PROGRAM Callblocks
VAR
	
Temp_bool : BOOL;
Mode_0          : Mode;
Feedback_FD     : Feedback_FB;
Feedback_RD     : Feedback_FB;
Feedback_FX1TR  : Feedback_FB;
Feedback_FX2TR  : Feedback_FB;
Feedback_TT     : Feedback_FB;
Feedback_CL     : Feedback_FB;

Front_Door        : RollerDoor;
Rear_Door         : RollerDoor;
Fixture1_Trunion  : Trunion;
Fixture2_Trunion  : Trunion;
TT                : Turntable ;
Robot1            : Weldrobot;
Robot2            : Weldrobot;



	
	MHRobot_0: MHRobot;
END_VAR

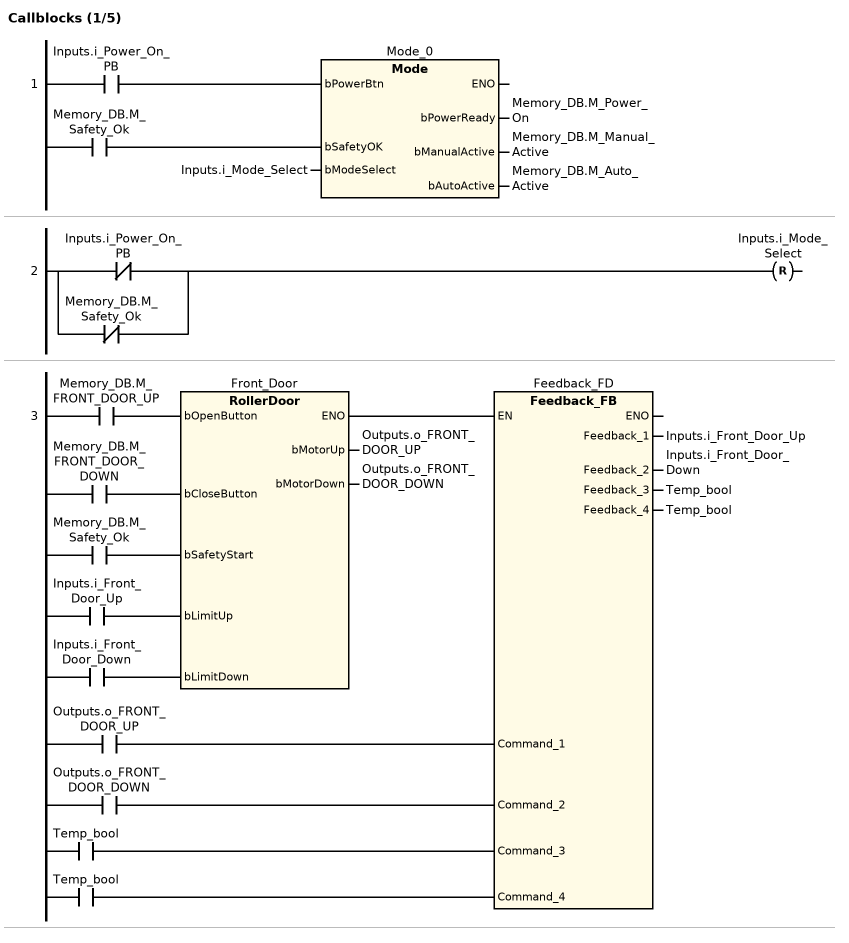
// NETWORK 1
Mode_0(
    bPowerBtn := Inputs.i_Power_On_PB,
    bSafetyOK := Memory_DB.M_Safety_Ok,
    bModeSelect := Inputs.i_Mode_Select,
    bPowerReady => Memory_DB.M_Power_On,
    bManualActive => Memory_DB.M_Manual_Active,
    bAutoActive => Memory_DB.M_Auto_Active); // Mode

// NETWORK 2
Inputs.i_Mode_Select R= NOT Inputs.i_Power_On_PB OR NOT Memory_DB.M_Safety_Ok;

// NETWORK 3
Front_Door(
    bOpenButton := Memory_DB.M_FRONT_DOOR_UP,
    bCloseButton := Memory_DB.M_FRONT_DOOR_DOWN,
    bSafetyStart := Memory_DB.M_Safety_Ok,
    bLimitUp := Inputs.i_Front_Door_Up,
    bLimitDown := Inputs.i_Front_Door_Down,
    bMotorUp => Outputs.o_FRONT_DOOR_UP,
    bMotorDown => Outputs.o_FRONT_DOOR_DOWN); // RollerDoor
Feedback_FD(
    EN := TRUE,
    Command_1 := Outputs.o_FRONT_DOOR_UP,
    Command_2 := Outputs.o_FRONT_DOOR_DOWN,
    Command_3 := Temp_bool,
    Command_4 := Temp_bool,
    Feedback_1 => Inputs.i_Front_Door_Up,
    Feedback_2 => Inputs.i_Front_Door_Down,
    Feedback_3 => Temp_bool,
    Feedback_4 => Temp_bool); // Feedback_FB

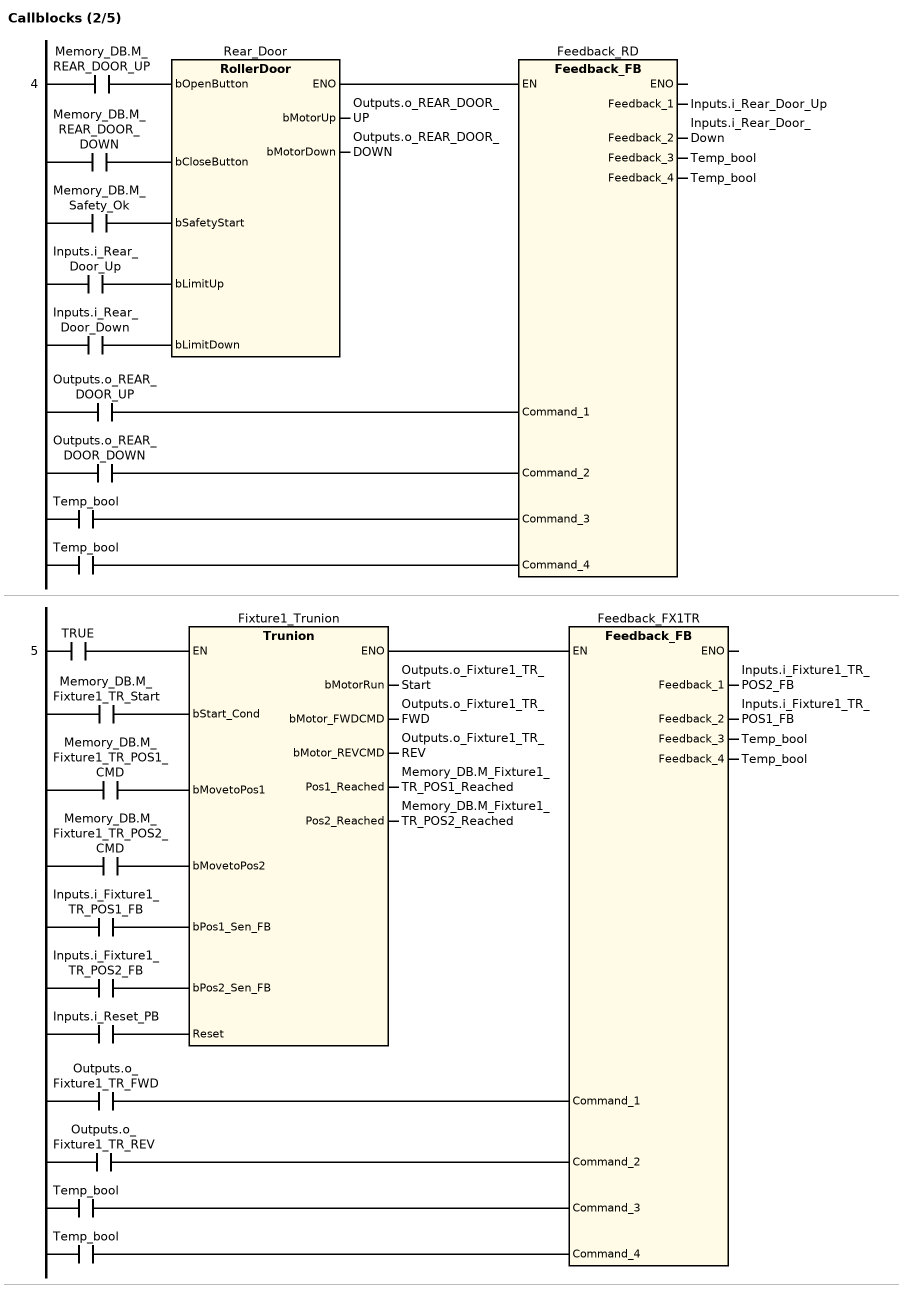
// NETWORK 4
Rear_Door(
    bOpenButton := Memory_DB.M_REAR_DOOR_UP,
    bCloseButton := Memory_DB.M_REAR_DOOR_DOWN,
    bSafetyStart := Memory_DB.M_Safety_Ok,
    bLimitUp := Inputs.i_Rear_Door_Up,
    bLimitDown := Inputs.i_Rear_Door_Down,
    bMotorUp => Outputs.o_REAR_DOOR_UP,
    bMotorDown => Outputs.o_REAR_DOOR_DOWN); // RollerDoor
Feedback_RD(
    EN := TRUE,
    Command_1 := Outputs.o_REAR_DOOR_UP,
    Command_2 := Outputs.o_REAR_DOOR_DOWN,
    Command_3 := Temp_bool,
    Command_4 := Temp_bool,
    Feedback_1 => Inputs.i_Rear_Door_Up,
    Feedback_2 => Inputs.i_Rear_Door_Down,
    Feedback_3 => Temp_bool,
    Feedback_4 => Temp_bool); // Feedback_FB

// NETWORK 5
Fixture1_Trunion(
    EN := TRUE,
    bStart_Cond := Memory_DB.M_Fixture1_TR_Start,
    bMovetoPos1 := Memory_DB.M_Fixture1_TR_POS1_CMD,
    bMovetoPos2 := Memory_DB.M_Fixture1_TR_POS2_CMD,
    bPos1_Sen_FB := Inputs.i_Fixture1_TR_POS1_FB,
    bPos2_Sen_FB := Inputs.i_Fixture1_TR_POS2_FB,
    Reset := Inputs.i_Reset_PB,
    bMotorRun => Outputs.o_Fixture1_TR_Start,
    bMotor_FWDCMD => Outputs.o_Fixture1_TR_FWD,
    bMotor_REVCMD => Outputs.o_Fixture1_TR_REV,
    Pos1_Reached => Memory_DB.M_Fixture1_TR_POS1_Reached,
    Pos2_Reached => Memory_DB.M_Fixture1_TR_POS2_Reached); // Trunion
Feedback_FX1TR(
    EN := TRUE,
    Command_1 := Outputs.o_Fixture1_TR_FWD,
    Command_2 := Outputs.o_Fixture1_TR_REV,
    Command_3 := Temp_bool,
    Command_4 := Temp_bool,
    Feedback_1 => Inputs.i_Fixture1_TR_POS2_FB,
    Feedback_2 => Inputs.i_Fixture1_TR_POS1_FB,
    Feedback_3 => Temp_bool,
    Feedback_4 => Temp_bool); // Feedback_FB

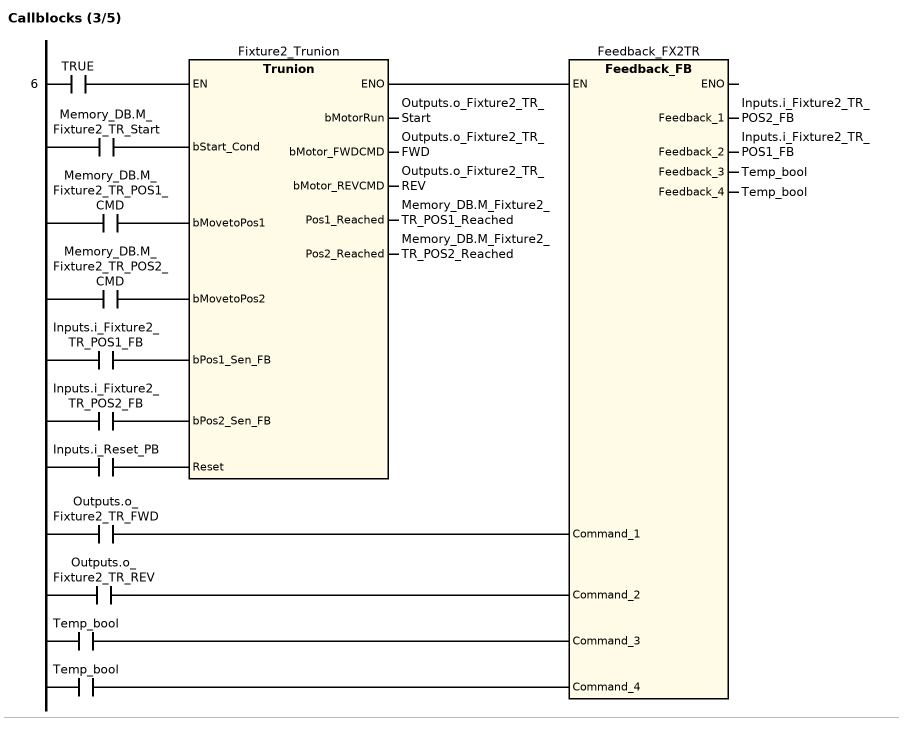
// NETWORK 6
Fixture2_Trunion(
    EN := TRUE,
    bStart_Cond := Memory_DB.M_Fixture2_TR_Start,
    bMovetoPos1 := Memory_DB.M_Fixture2_TR_POS1_CMD,
    bMovetoPos2 := Memory_DB.M_Fixture2_TR_POS2_CMD,
    bPos1_Sen_FB := Inputs.i_Fixture2_TR_POS1_FB,
    bPos2_Sen_FB := Inputs.i_Fixture2_TR_POS2_FB,
    Reset := Inputs.i_Reset_PB,
    bMotorRun => Outputs.o_Fixture2_TR_Start,
    bMotor_FWDCMD => Outputs.o_Fixture2_TR_FWD,
    bMotor_REVCMD => Outputs.o_Fixture2_TR_REV,
    Pos1_Reached => Memory_DB.M_Fixture2_TR_POS1_Reached,
    Pos2_Reached => Memory_DB.M_Fixture2_TR_POS2_Reached); // Trunion
Feedback_FX2TR(
    EN := TRUE,
    Command_1 := Outputs.o_Fixture2_TR_FWD,
    Command_2 := Outputs.o_Fixture2_TR_REV,
    Command_3 := Temp_bool,
    Command_4 := Temp_bool,
    Feedback_1 => Inputs.i_Fixture2_TR_POS2_FB,
    Feedback_2 => Inputs.i_Fixture2_TR_POS1_FB,
    Feedback_3 => Temp_bool,
    Feedback_4 => Temp_bool); // Feedback_FB

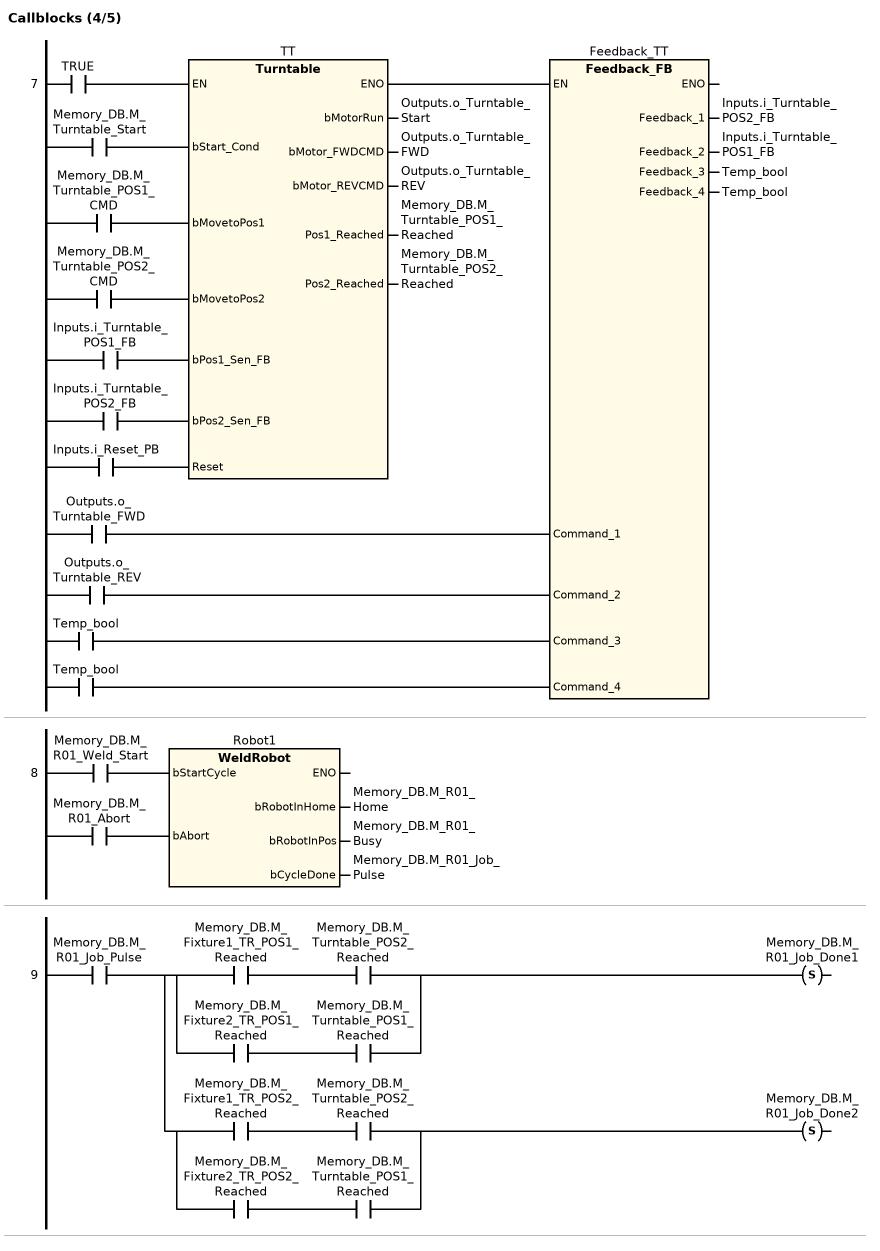
// NETWORK 7
TT(
    EN := TRUE,
    bStart_Cond := Memory_DB.M_Turntable_Start,
    bMovetoPos1 := Memory_DB.M_Turntable_POS1_CMD,
    bMovetoPos2 := Memory_DB.M_Turntable_POS2_CMD,
    bPos1_Sen_FB := Inputs.i_Turntable_POS1_FB,
    bPos2_Sen_FB := Inputs.i_Turntable_POS2_FB,
    Reset := Inputs.i_Reset_PB,
    bMotorRun => Outputs.o_Turntable_Start,
    bMotor_FWDCMD => Outputs.o_Turntable_FWD,
    bMotor_REVCMD => Outputs.o_Turntable_REV,
    Pos1_Reached => Memory_DB.M_Turntable_POS1_Reached,
    Pos2_Reached => Memory_DB.M_Turntable_POS2_Reached); // Turntable
Feedback_TT(
    EN := TRUE,
    Command_1 := Outputs.o_Turntable_FWD,
    Command_2 := Outputs.o_Turntable_REV,
    Command_3 := Temp_bool,
    Command_4 := Temp_bool,
    Feedback_1 => Inputs.i_Turntable_POS2_FB,
    Feedback_2 => Inputs.i_Turntable_POS1_FB,
    Feedback_3 => Temp_bool,
    Feedback_4 => Temp_bool); // Feedback_FB

// NETWORK 8
Robot1(
    bStartCycle := Memory_DB.M_R01_Weld_Start,
    bAbort := Memory_DB.M_R01_Abort,
    bRobotInHome => Memory_DB.M_R01_Home,
    bRobotInPos => Memory_DB.M_R01_Busy,
    bCycleDone => Memory_DB.M_R01_Job_Pulse); // WeldRobot

// NETWORK 9
Memory_DB.M_R01_Job_Done1 S= (Memory_DB.M_R01_Job_Pulse AND Memory_DB.M_Fixture1_TR_POS1_Reached) AND Memory_DB.M_Turntable_POS2_Reached OR (Memory_DB.M_R01_Job_Pulse AND Memory_DB.M_Fixture2_TR_POS1_Reached) AND Memory_DB.M_Turntable_POS1_Reached;
Memory_DB.M_R01_Job_Done2 S= (Memory_DB.M_R01_Job_Pulse AND Memory_DB.M_Fixture1_TR_POS2_Reached) AND Memory_DB.M_Turntable_POS2_Reached OR (Memory_DB.M_R01_Job_Pulse AND Memory_DB.M_Fixture2_TR_POS2_Reached) AND Memory_DB.M_Turntable_POS1_Reached;

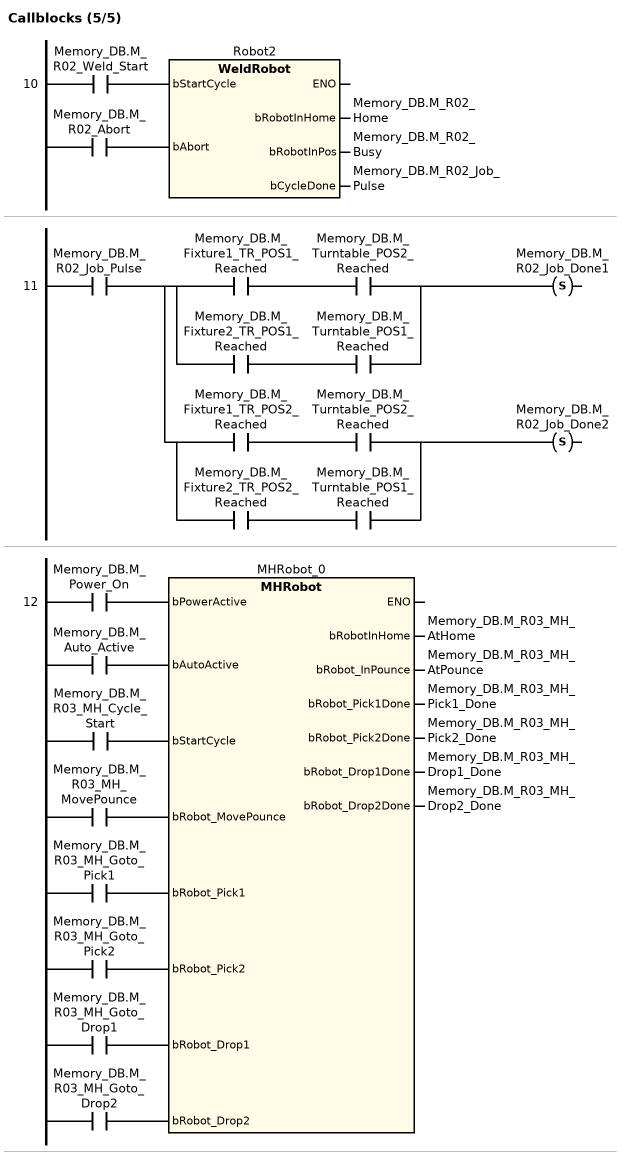
// NETWORK 10
Robot2(
    bStartCycle := Memory_DB.M_R02_Weld_Start,
    bAbort := Memory_DB.M_R02_Abort,
    bRobotInHome => Memory_DB.M_R02_Home,
    bRobotInPos => Memory_DB.M_R02_Busy,
    bCycleDone => Memory_DB.M_R02_Job_Pulse); // WeldRobot

// NETWORK 11
Memory_DB.M_R02_Job_Done1 S= (Memory_DB.M_R02_Job_Pulse AND Memory_DB.M_Fixture1_TR_POS1_Reached) AND Memory_DB.M_Turntable_POS2_Reached OR (Memory_DB.M_R02_Job_Pulse AND Memory_DB.M_Fixture2_TR_POS1_Reached) AND Memory_DB.M_Turntable_POS1_Reached;
Memory_DB.M_R02_Job_Done2 S= (Memory_DB.M_R02_Job_Pulse AND Memory_DB.M_Fixture1_TR_POS2_Reached) AND Memory_DB.M_Turntable_POS2_Reached OR (Memory_DB.M_R02_Job_Pulse AND Memory_DB.M_Fixture2_TR_POS2_Reached) AND Memory_DB.M_Turntable_POS1_Reached;

// NETWORK 12
MHRobot_0(
    bPowerActive := Memory_DB.M_Power_On,
    bAutoActive := Memory_DB.M_Auto_Active,
    bStartCycle := Memory_DB.M_R03_MH_Cycle_Start,
    bRobot_MovePounce := Memory_DB.M_R03_MH_MovePounce,
    bRobot_Pick1 := Memory_DB.M_R03_MH_Goto_Pick1,
    bRobot_Pick2 := Memory_DB.M_R03_MH_Goto_Pick2,
    bRobot_Drop1 := Memory_DB.M_R03_MH_Goto_Drop1,
    bRobot_Drop2 := Memory_DB.M_R03_MH_Goto_Drop2,
    bRobotInHome => Memory_DB.M_R03_MH_AtHome,
    bRobot_InPounce => Memory_DB.M_R03_MH_AtPounce,
    bRobot_Pick1Done => Memory_DB.M_R03_MH_Pick1_Done,
    bRobot_Pick2Done => Memory_DB.M_R03_MH_Pick2_Done,
    bRobot_Drop1Done => Memory_DB.M_R03_MH_Drop1_Done,
    bRobot_Drop2Done => Memory_DB.M_R03_MH_Drop2_Done); // MHRobot

END_PROGRAM

(* stored: Version 1.1.0.1, ProductVersion 3.1.4024.16
   POU Callblocks: Id {48d0d7d2-3848-41ce-8b0c-24cedca1c020}, SpecialFunc None *)
